(* Schneider Machine Expert - Basic project FlandersHVL_V2, file version 1.8.0.0 *)
(* ProjectInformations: Name=New project *)

HARDWARE
  Cpu 0: TM221CE24R
  ModuleExtensionObject 0: TM3AQ4/G
  ModuleExtensionObject 1: TM2DDO8TT
  EthernetConfiguration: NetworkName=M221, IpAllocationMode=FixedAddress, IpAddress=0.0.0.0, SubnetMask=0.0.0.0
  SerialLineConfiguration: Baud=Baud19200, Parity=ParityEven, DataBits=DataBits8, StopBits=StopBits1, PhysicalMedium=PhysicalMediumRs485, TransmissionMode=TransmissionModeModbusRtu, SlaveId=1, Addressing=SlaveAddressing
  MastTask: UsePeriodScanMode=false, PeriodScan=100
  FastTask: Period=255
  CpuBehavior: StartingMode=StartAsPreviousState, AutoSaveRamOnEeprom=true, WatchdogPeriod=250

SYMBOLS  (address, symbol, comment, settings)
  %M0       RESET
  %M1       RUN_STRIP_PULL_CYCLE
  %M2       EXTEND_CLAMP
  %M3       GLUE_TIMER_DN
  %M4       RUN_GLUE_CYCLE
  %M5       SYSTEM_RUNNING
  %M6       MCR  "Master Control Relay"
  %M7       SYSTEM_IDLE
  %M8       SYSTEM_START
  %M9       PHYSICAL_ALARM_TIMEOUT
  %M10      SYNC_STRIPS
  %M11      ONE_MIN_PASSED
  %M12      NEXT_SPEED
  %M13      START_RPM_TEST
  %M14      STRIP_PULL_STEP_1
  %M15      STRIP_PULL_LAST_STEP
  %M16      SYNC_VACS
  %M17      SYNC_STRIP_CYL_OUT
  %M18      SYN_STRIP_CYL_IN
  %M19      SYNC_PINS
  %M20      SYNC_GLUE
  %M21      SYNC_STRIP_MOTORS
  %M100     TEST_BIT
  %TM0      STOP_ALARM_TIMER
  %TM1      GLUE_TIMER  "Used to make sure glue doesn't go off the edge of the strip"
  %TM2      FPM_SPEED_TIMER  [Base=TenMilliSeconds]
  %TM3      MEDIA_DETECT_TIMER  [Preset=700, Base=OneMilliSeconds]
  %TM4      VAC_ON_DELAY  [Preset=1, Base=OneSecond]
  %C0       FILTER_PER_MINUTE_COUNTER
  %I0.0     SPEED_DETECT
  %I0.1     FLIGHT_DETECT
  %I0.2     VAC_CYL_A_OUT
  %I0.3     VAC_CYL_A_IN
  %I0.4     VAC_CYL_B_OUT
  %I0.5     VAC_CYL_B_IN
  %I0.6     MEDIA_DETECT
  %I0.7     STRIP_DETECT_A
  %I0.8     STRIP_DETECT_B
  %I0.9     GLUE_EYE
  %I0.10    SAFETY
  %Q0.0     VAC_A
  %Q0.1     VAC_B
  %Q0.2     STRIP_A
  %Q0.3     STRIP_B
  %Q0.4     PIN_A
  %Q0.5     PIN_B
  %Q0.6     GLUE_HEAD_A_TOP
  %Q0.7     GLUE_HEAD_A_BOT
  %Q0.8     GLUE_HEAD_B_TOP
  %Q0.9     GLUE_HEAD_B_BOT
  %QW1.0    DRIVE_MOTOR  [Type=Type_0_10V, Scope=Scope_Customized, Minimum=0, Maximum=10000]
  %Q2.0     PHYSICAL_ALARM
  %Q2.3     PINCH_ROLLER_MOTOR
  %Q2.4     STRIP_B_MOTOR
  %Q2.5     STRIP_A_MOTOR

POU Strip_Machine
  (* SectionNumber=1 *)

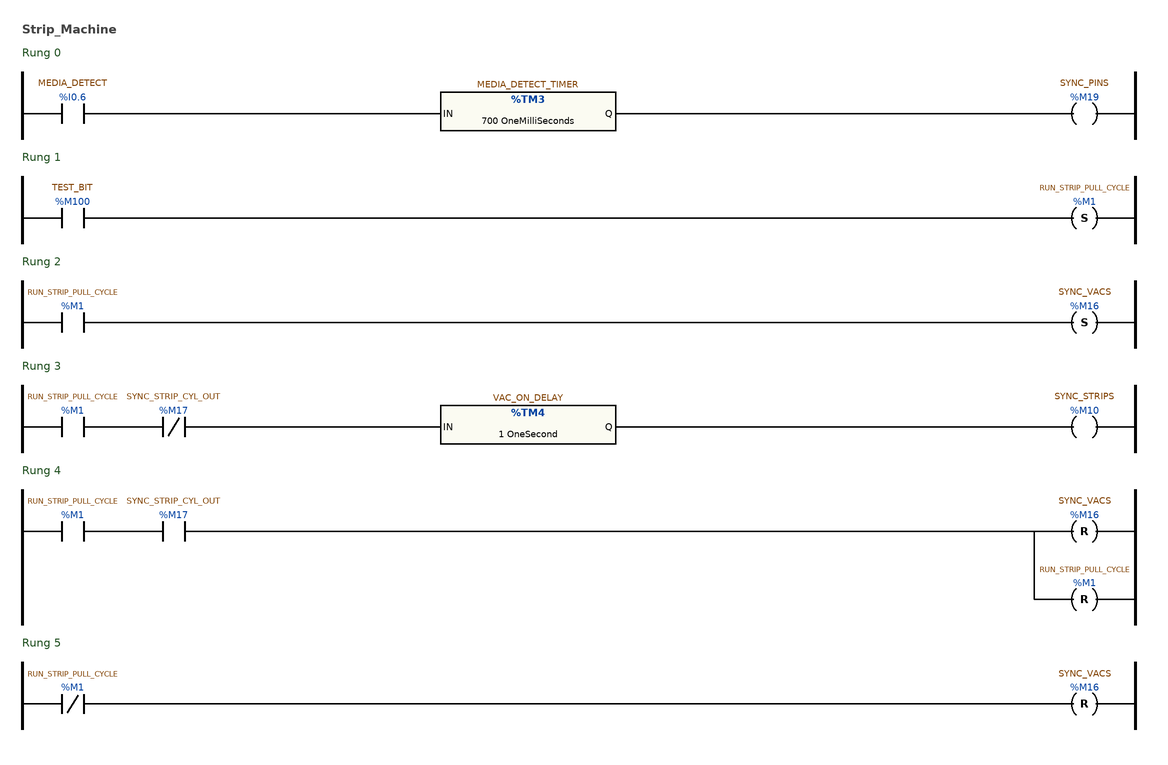

// Rung 0
  BLK %TM3                (* MEDIA_DETECT_TIMER *)
  LD %I0.6                (* MEDIA_DETECT *)
  IN
  OUT_BLK
  LD Q
  ST %M19                 (* SYNC_PINS *)
  END_BLK
  // as ST:
  //   MEDIA_DETECT_TIMER(IN := MEDIA_DETECT);
  //   SYNC_PINS := MEDIA_DETECT_TIMER.Q;

// Rung 1
  LD %M100                (* TEST_BIT *)
  S %M1                   (* RUN_STRIP_PULL_CYCLE *)
  // as ST:
  //   IF TEST_BIT THEN RUN_STRIP_PULL_CYCLE := TRUE; END_IF;

// Rung 2
  LD %M1                  (* RUN_STRIP_PULL_CYCLE *)
  S %M16                  (* SYNC_VACS *)
  // as ST:
  //   IF RUN_STRIP_PULL_CYCLE THEN SYNC_VACS := TRUE; END_IF;

// Rung 3
  BLK %TM4                (* VAC_ON_DELAY *)
  LD %M1                  (* RUN_STRIP_PULL_CYCLE *)
  ANDN %M17               (* SYNC_STRIP_CYL_OUT *)
  IN
  OUT_BLK
  LD Q
  ST %M10                 (* SYNC_STRIPS *)
  END_BLK
  // as ST:
  //   VAC_ON_DELAY(IN := RUN_STRIP_PULL_CYCLE AND NOT SYNC_STRIP_CYL_OUT);
  //   SYNC_STRIPS := VAC_ON_DELAY.Q;

// Rung 4
  LD %M1                  (* RUN_STRIP_PULL_CYCLE *)
  AND %M17                (* SYNC_STRIP_CYL_OUT *)
  R %M16                  (* SYNC_VACS *)
  R %M1                   (* RUN_STRIP_PULL_CYCLE *)
  // as ST:
  //   IF RUN_STRIP_PULL_CYCLE AND SYNC_STRIP_CYL_OUT THEN SYNC_VACS := FALSE; END_IF;
  //   IF RUN_STRIP_PULL_CYCLE AND SYNC_STRIP_CYL_OUT THEN RUN_STRIP_PULL_CYCLE := FALSE; END_IF;

// Rung 5
  LDN %M1                 (* RUN_STRIP_PULL_CYCLE *)
  R %M16                  (* SYNC_VACS *)
  // as ST:
  //   IF NOT RUN_STRIP_PULL_CYCLE THEN SYNC_VACS := FALSE; END_IF;

POU High_Power_Devices
  (* SectionNumber=2 *)

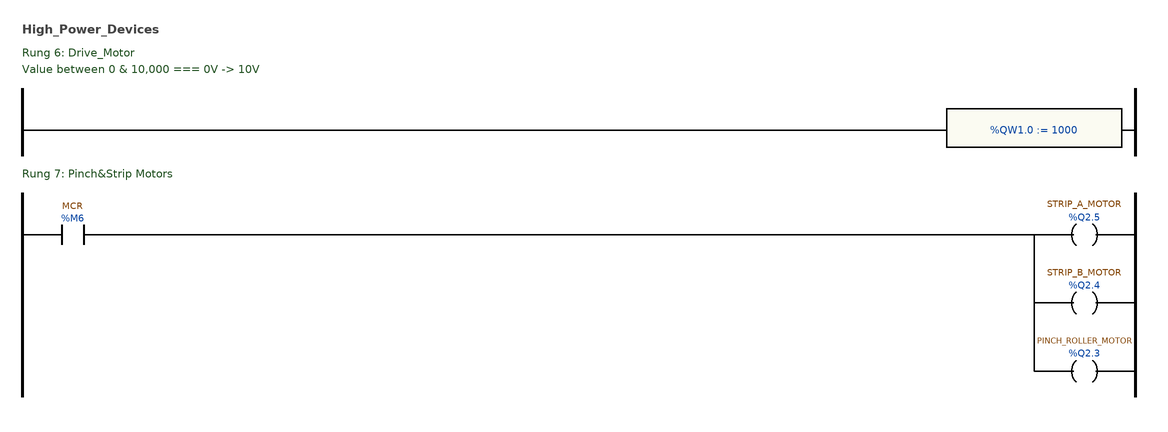

// Rung 6: Drive_Motor
// Value between 0 & 10,000 === 0V -> 10V
  LD 1
  [ %QW1.0 := 1000 ]      (* DRIVE_MOTOR *)
  // as ST:
  //   DRIVE_MOTOR := 1000;

// Rung 7: Pinch&Strip Motors
  LD %M6                  (* MCR *)
  ST %Q2.5                (* STRIP_A_MOTOR *)
  ST %Q2.4                (* STRIP_B_MOTOR *)
  ST %Q2.3                (* PINCH_ROLLER_MOTOR *)
  // as ST:
  //   STRIP_A_MOTOR := MCR;
  //   STRIP_B_MOTOR := MCR;
  //   PINCH_ROLLER_MOTOR := MCR;

POU RPM
  (* SectionNumber=3 *)

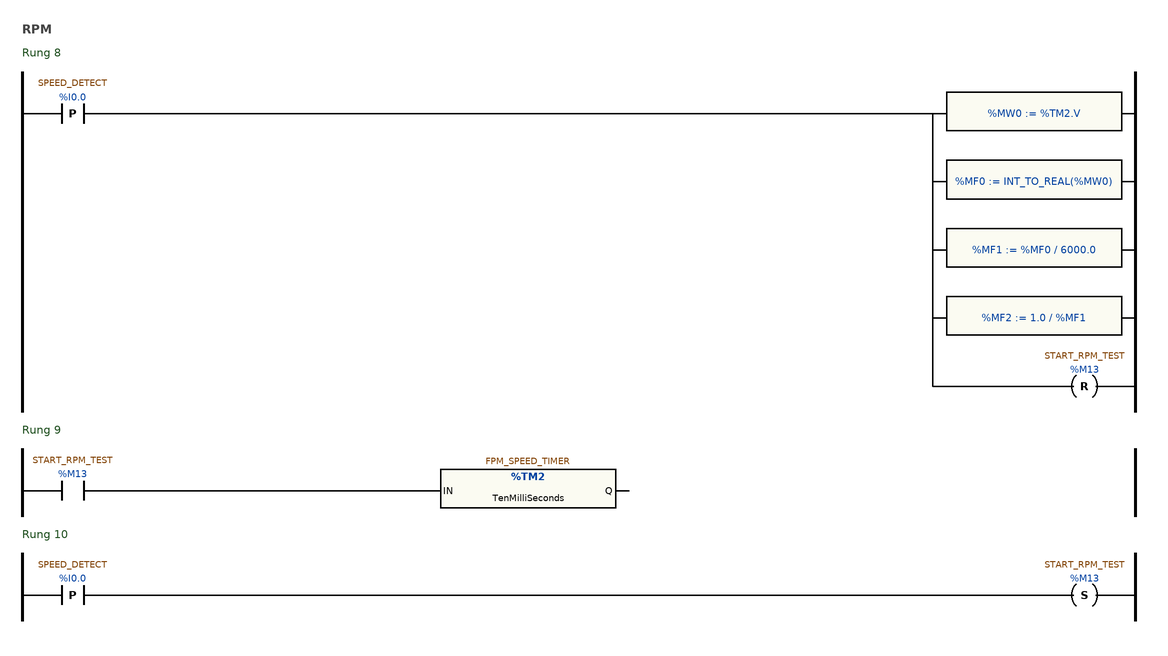

// Rung 8
  LDR %I0.0               (* SPEED_DETECT *)
  [ %MW0 := %TM2.V ]      (* FPM_SPEED_TIMER *)
  [ %MF0 := INT_TO_REAL ( %MW0 ) ]
  [ %MF1 := %MF0 / 6000.0 ]
  [ %MF2 := 1.0 / %MF1 ]
  R %M13                  (* START_RPM_TEST *)
  // as ST:
  //   IF RISING(SPEED_DETECT) THEN %MW0 := FPM_SPEED_TIMER.V; END_IF;
  //   IF RISING(SPEED_DETECT) THEN %MF0 := INT_TO_REAL ( %MW0 ); END_IF;
  //   IF RISING(SPEED_DETECT) THEN %MF1 := %MF0  /  6000.0; END_IF;
  //   IF RISING(SPEED_DETECT) THEN %MF2 := 1.0  /  %MF1; END_IF;
  //   IF RISING(SPEED_DETECT) THEN START_RPM_TEST := FALSE; END_IF;

// Rung 9
  BLK %TM2                (* FPM_SPEED_TIMER *)
  LD %M13                 (* START_RPM_TEST *)
  IN
  END_BLK
  // as ST:
  //   FPM_SPEED_TIMER(IN := START_RPM_TEST);

// Rung 10
  LDR %I0.0               (* SPEED_DETECT *)
  S %M13                  (* START_RPM_TEST *)
  // as ST:
  //   IF RISING(SPEED_DETECT) THEN START_RPM_TEST := TRUE; END_IF;

POU Synchronize
  (* SectionNumber=4 *)

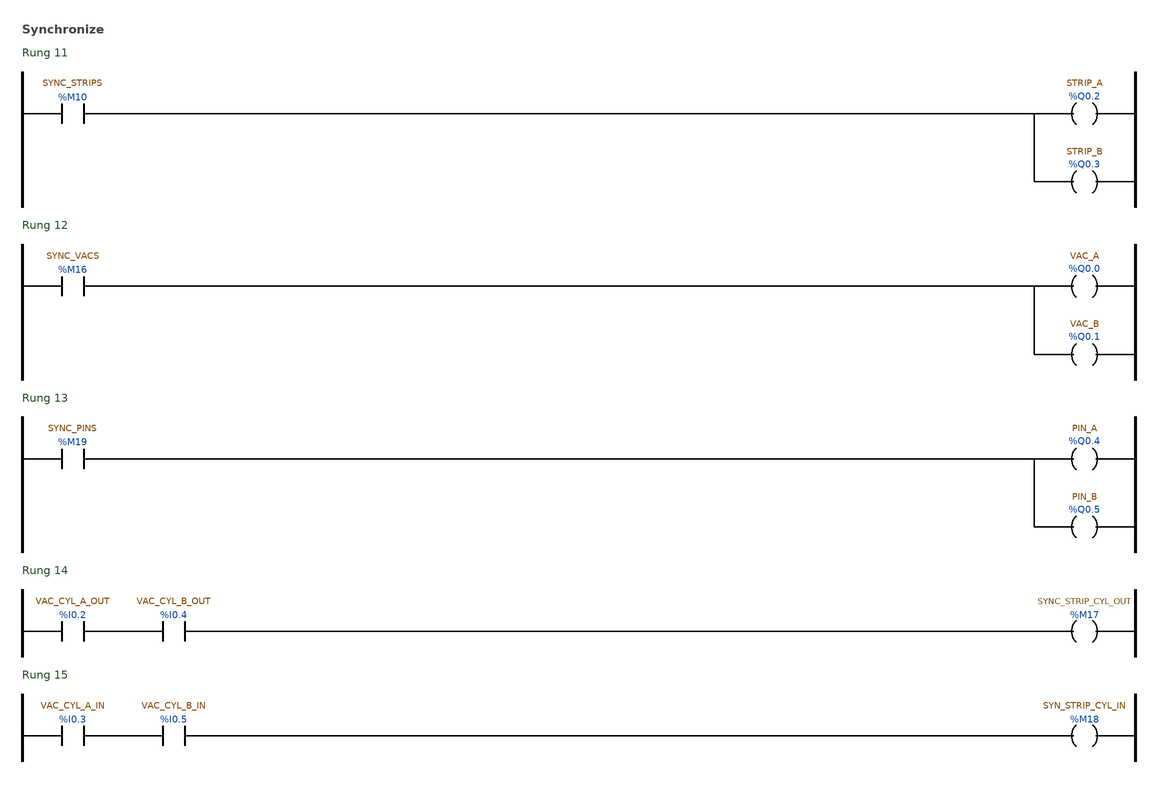

// Rung 11
  LD %M10                 (* SYNC_STRIPS *)
  ST %Q0.2                (* STRIP_A *)
  ST %Q0.3                (* STRIP_B *)
  // as ST:
  //   STRIP_A := SYNC_STRIPS;
  //   STRIP_B := SYNC_STRIPS;

// Rung 12
  LD %M16                 (* SYNC_VACS *)
  ST %Q0.0                (* VAC_A *)
  ST %Q0.1                (* VAC_B *)
  // as ST:
  //   VAC_A := SYNC_VACS;
  //   VAC_B := SYNC_VACS;

// Rung 13
  LD %M19                 (* SYNC_PINS *)
  ST %Q0.4                (* PIN_A *)
  ST %Q0.5                (* PIN_B *)
  // as ST:
  //   PIN_A := SYNC_PINS;
  //   PIN_B := SYNC_PINS;

// Rung 14
  LD %I0.2                (* VAC_CYL_A_OUT *)
  AND %I0.4               (* VAC_CYL_B_OUT *)
  ST %M17                 (* SYNC_STRIP_CYL_OUT *)
  // as ST:
  //   SYNC_STRIP_CYL_OUT := VAC_CYL_A_OUT AND VAC_CYL_B_OUT;

// Rung 15
  LD %I0.3                (* VAC_CYL_A_IN *)
  AND %I0.5               (* VAC_CYL_B_IN *)
  ST %M18                 (* SYN_STRIP_CYL_IN *)
  // as ST:
  //   SYN_STRIP_CYL_IN := VAC_CYL_A_IN AND VAC_CYL_B_IN;

POU Sytem Signals
  (* SectionNumber=5 *)

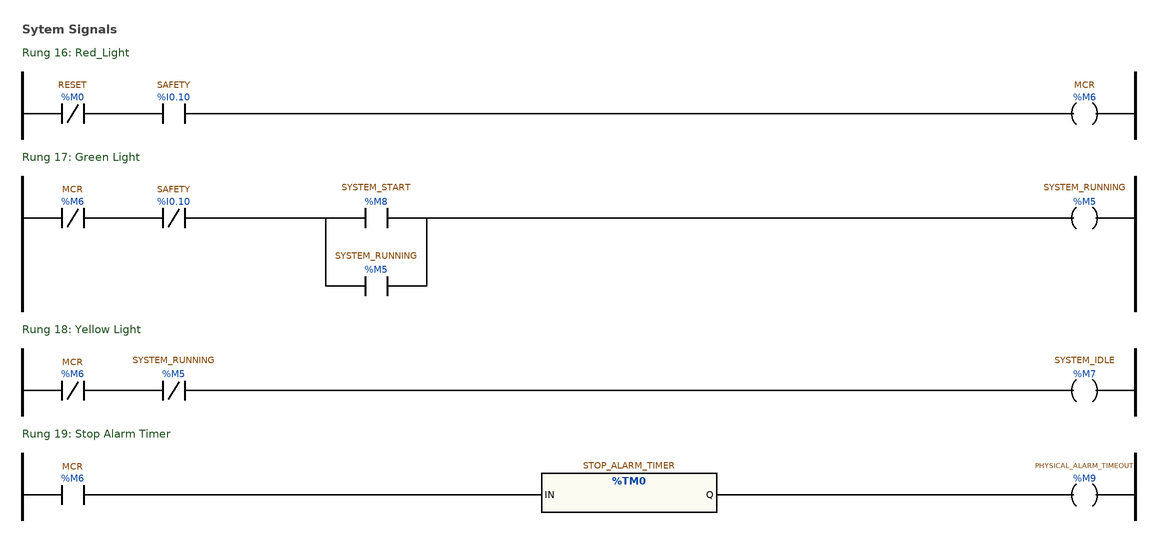

// Rung 16: Red_Light
  LDN %M0                 (* RESET *)
  AND %I0.10              (* SAFETY *)
  ST %M6                  (* MCR *)
  // as ST:
  //   MCR := NOT RESET AND SAFETY;

// Rung 17: Green Light
  LDN %M6                 (* MCR *)
  ANDN %I0.10             (* SAFETY *)
  AND( %M8                (* SYSTEM_START *)
  OR %M5                  (* SYSTEM_RUNNING *)
  )
  ST %M5                  (* SYSTEM_RUNNING *)
  // as ST:
  //   SYSTEM_RUNNING := NOT MCR AND NOT SAFETY AND (SYSTEM_START OR SYSTEM_RUNNING);

// Rung 18: Yellow Light
  LDN %M6                 (* MCR *)
  ANDN %M5                (* SYSTEM_RUNNING *)
  ST %M7                  (* SYSTEM_IDLE *)
  // as ST:
  //   SYSTEM_IDLE := NOT MCR AND NOT SYSTEM_RUNNING;

// Rung 19: Stop Alarm Timer
  BLK %TM0                (* STOP_ALARM_TIMER *)
  LD %M6                  (* MCR *)
  IN
  OUT_BLK
  LD Q
  ST %M9                  (* PHYSICAL_ALARM_TIMEOUT *)
  END_BLK
  // as ST:
  //   STOP_ALARM_TIMER(IN := MCR);
  //   PHYSICAL_ALARM_TIMEOUT := STOP_ALARM_TIMER.Q;
